# EPICS IOC start-up script: hugo/source/examples/test/PSI/ep2308.iocsh
#- #############################################################################
#- mXsXXX naming
require ecmccfg v7_RC1, "NAMING=mXsXXX"

#- #############################################################################
#- add slaves
${SCRIPTEXEC} ${ecmccfg_DIR}addSlave.cmd, "HW_DESC=EP2308, SLAVE_ID=${SLAVE=5}"

#- #############################################################################
#- apply hardware configuration
${SCRIPTEXEC} ${ecmccfg_DIR}applyConfig.cmd

#- #############################################################################
#- configure diagnostics
ecmcConfigOrDie "Cfg.EcSetDiagnostics(1)"
ecmcConfigOrDie "Cfg.EcEnablePrintouts(0)"
ecmcConfigOrDie "Cfg.EcSetDomainFailedCyclesLimit(100)"

# go active
${SCRIPTEXEC} ${ecmccfg_DIR}setAppMode.cmd
#- #############################################################################
